FUNCTION_BLOCK Motor_Direction
VAR_INPUT
	startMove: BOOL;
	currentPositon: UINT;
	desiredPositon: UINT;
	refLimitSwitch: BOOL;
	positveMove: BOOL;
	negativeMove: BOOL;
	tolerance: UINT;
	enableCounterWrite: BOOL;
	desiredSpeed: INT;
	//setEncoder: UINT;
	
END_VAR
VAR_OUTPUT
	setPositveMove: BOOL;
	setNegativeMove: BOOL;
	setPositionCounter: UINT;
	setEnable: INT;
	setSpeedPWM:INT;
END_VAR
VAR
	referencePosition: UINT :=0;
	
	motorEnable_vertival: Motor_Enable;
END_VAR

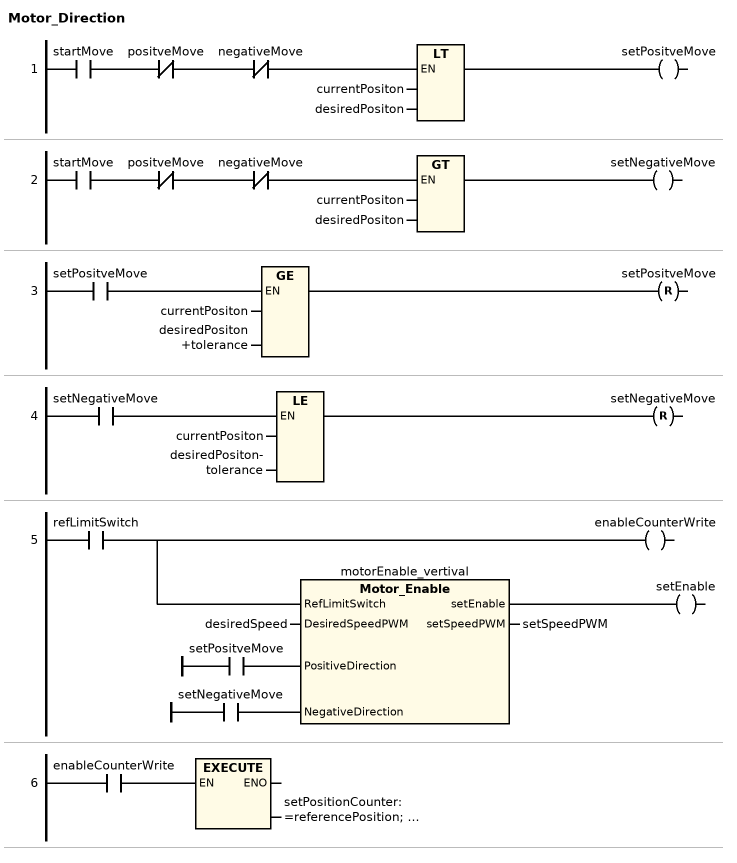
// NETWORK 1
setPositveMove := startMove AND NOT positveMove AND NOT negativeMove AND currentPositon < desiredPositon;

// NETWORK 2
setNegativeMove := startMove AND NOT positveMove AND NOT negativeMove AND currentPositon > desiredPositon;

// NETWORK 3
setPositveMove R= setPositveMove AND currentPositon >= (desiredPositon +tolerance);

// NETWORK 4
setNegativeMove R= setNegativeMove AND currentPositon <= (desiredPositon-tolerance);

// NETWORK 5
enableCounterWrite := refLimitSwitch;
motorEnable_vertival(
    RefLimitSwitch := refLimitSwitch,
    DesiredSpeedPWM := desiredSpeed,
    PositiveDirection := setPositveMove,
    NegativeDirection := setNegativeMove,
    setSpeedPWM => setSpeedPWM); // Motor_Enable
setEnable := motorEnable_vertival.setEnable;

// NETWORK 6
IF enableCounterWrite THEN setPositionCounter:=referencePosition; END_IF

END_FUNCTION_BLOCK

(* stored: Version 1.1.0.1, ProductVersion 3.1.4024.12
   POU Motor_Direction: Id {8fbc4570-101c-4e39-9754-c7aafbc7da5f}, SpecialFunc None *)
